(* PLC project Tc3_EventLogger.OnAlarmCleared Demo, tc3-libraries-kb TwinCAT 3.1 *)
(* stored: creationDateTime 2026-05-11T01:00:00, modificationDateTime 2026-05-11T01:00:00 *)

PROGRAM P_Demo_OnAlarmCleared
  VAR
    fbOnAlarmCleared : OnAlarmCleared;  (* Tc3_EventLogger.OnAlarmCleared 实例 *)
    arg_fbEvent : REFERENCE TO FB_TcEvent;  (* VAR_INPUT fbEvent *)
  END_VAR

            // ============================================================
// Tc3_EventLogger.OnAlarmCleared 演示程序（FB 实例）
// ============================================================
// 验证步骤：
//   1. 引用 Tc3_EventLogger（及依赖类型所在库 Tc2_System 等）
//   2. 编译 + 登录
//   3. 按 doc.md 给 arg_* 赋值
//   4. 在线监视 out_* / io_* 输出
// ============================================================

fbOnAlarmCleared(
    fbEvent := arg_fbEvent
);

          
END_PROGRAM
